(* PLC project VendorAddDataFixture, RoboC++ Validation Vendor AddData Fixture 1.0 *)
(* stored: creationDateTime 2026-05-29T00:00:00, modificationDateTime 2026-05-29T00:00:00 *)

PROGRAM VendorAddDataProgram
  VAR
    A : INT;
  END_VAR

            A := A + 1;
          
END_PROGRAM
